FUNCTION_BLOCK C_HTTP_BASE
VAR_INPUT
END_VAR
VAR_OUTPUT
END_VAR
VAR
END_VAR

PROPERTY Line_Space : String(1)
GET
Line_Space := ' ';
END_GET
END_PROPERTY

PROPERTY Line_Terminator : STRING(2)
GET
Line_Terminator := '$R$N';
END_GET
END_PROPERTY

PROPERTY PROTECTED Url_Split_Charactor : STRING(1)
GET
Url_Split_Charactor := '/';
END_GET
END_PROPERTY

END_FUNCTION_BLOCK

(* stored: Version 1.1.0.1, ProductVersion 3.1.4019.2
   POU C_HTTP_BASE: Id {12de8f6a-11e0-44df-8e22-77dc018836cb}, SpecialFunc None
   Property Line_Space: Id {23e9f583-afef-4949-95f9-9b835024c173}
   Get Get: Id {f693bc7d-fa57-46de-b794-7017a3b7fa7f}
   Property Line_Terminator: Id {0fb95a2d-b8fb-44a1-9469-65cd5bfeb118}
   Get Get: Id {ef1f5196-8288-4220-871b-5b239b36612a}
   Property Url_Split_Charactor: Id {bcc3e33d-a2d4-419a-bea0-49952b86deec}
   Get Get: Id {a73ed253-cc19-4b50-9830-f2395f2dac63} *)
